// TIA Portal V18 export
DATA_BLOCK "CTRL_PWM_DB"   // DB32
// stored: AutoNumber true, DBAccessibleFromOPCUA true, InstanceOfName CTRL_PWM_SFB, OfSystemLibElement CTRL_PWM, OfSystemLibVersion 1.0
"CTRL_PWM_SFB"
   // VAR_INPUT
   //    PWM : HW_PWM;
   //    ENABLE : Bool;
   // END_VAR
   // VAR_OUTPUT
   //    BUSY : Bool;
   //    STATUS : Word;
   // END_VAR
BEGIN
END_DATA_BLOCK
